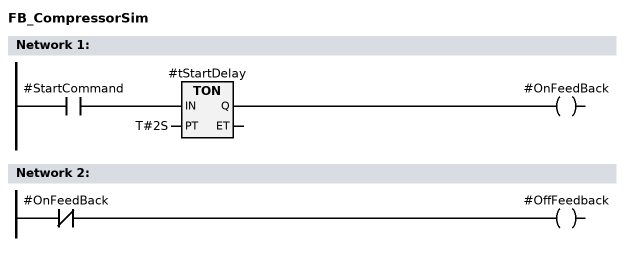
   #tStartDelay(IN := #StartCommand, PT := T#2S);   // TON
   #OnFeedBack := #tStartDelay.Q;
END_REGION

REGION Network 2
   RUNG wire#powerrail
      I_Contact( #OnFeedBack )
      Coil( #OffFeedback )
   END_RUNG
   // the same network as SCL:
   #OffFeedback := NOT #OnFeedBack;
END_REGION
END_FUNCTION_BLOCK

FUNCTION_BLOCK "FB_FanSim"   // FB9, LAD
{ S7_Optimized_Access := 'TRUE' }
VERSION : 0.1
   VAR_INPUT
      StartCommand : Bool;
   END_VAR
   VAR_OUTPUT
      OnFeedBack : Bool;
      OffFeedBack : Bool;
   END_VAR
   VAR
      tStartDelay : TON_TIME;
      SA : Bool;
   END_VAR
   VAR_TEMP
      Temp_1 : Bool;
   END_VAR
BEGIN

REGION Network 1
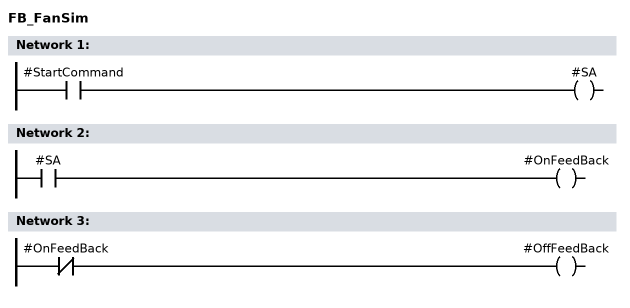
   RUNG wire#powerrail
      Contact( #StartCommand )
      Coil( #SA )
   END_RUNG
   // the same network as SCL:
   #SA := #StartCommand;
END_REGION

REGION Network 2
   RUNG wire#powerrail
      Contact( #SA )
      Coil( #OnFeedBack )
   END_RUNG
   // the same network as SCL:
   #OnFeedBack := #SA;
END_REGION

REGION Network 3
   RUNG wire#powerrail
      I_Contact( #OnFeedBack )
      Coil( #OffFeedBack )
   END_RUNG
   // the same network as SCL:
   #OffFeedBack := NOT #OnFeedBack;
END_REGION
END_FUNCTION_BLOCK

(* ===== HMI "HMI_RT_1" =====
system functions are stored by id; their names below are inferred from use
connection "HMI_Connection_1": ETHERNET, S7_1500_OMS

HMI tags "Default tag table"
   "Db_Equipment_Compressor{1}_Sts_Status" : Int = PLC Db_Equipment.Compressor[1].Sts.Status, 1 s
   "Db_Equipment_Compressor{2}_Sts_Status" : Int = PLC Db_Equipment.Compressor[2].Sts.Status, 1 s
   "Db_Equipment_Compressor{3}_Sts_Status" : Int = PLC Db_Equipment.Compressor[3].Sts.Status, 1 s
   "Db_Equipment_Compressor{4}_Sts_Status" : Int = PLC Db_Equipment.Compressor[4].Sts.Status, 1 s
   "Db_Equipment_Compressor{5}_Sts_Status" : Int = PLC Db_Equipment.Compressor[5].Sts.Status, 1 s
   "Db_Equipment_Compressor{6}_Sts_Status" : Int = PLC Db_Equipment.Compressor[6].Sts.Status, 1 s
   "Db_Equipment_Compressor{7}_Sts_Status" : Int = PLC Db_Equipment.Compressor[7].Sts.Status, 1 s
   "Db_Equipment_Compressor{8}_Sts_Status" : Int = PLC Db_Equipment.Compressor[8].Sts.Status, 1 s
   "Db_Equipment_Fan{1}_Sts_Status" : Int = PLC Db_Equipment.Fan[1].Sts.Status, 1 s
   "Db_Equipment_Fan{2}_Sts_Status" : Int = PLC Db_Equipment.Fan[2].Sts.Status, 1 s
   "Db_Equipment_Fan{3}_Sts_Status" : Int = PLC Db_Equipment.Fan[3].Sts.Status, 1 s
   "Db_Equipment_Fan{4}_Sts_Status" : Int = PLC Db_Equipment.Fan[4].Sts.Status, 1 s
   "Db_Equipment_Fan{5}_Sts_Status" : Int = PLC Db_Equipment.Fan[5].Sts.Status, 1 s
   "Db_Equipment_Fan{6}_Sts_Status" : Int = PLC Db_Equipment.Fan[6].Sts.Status, 1 s
   "Db_Equipment_Fan{7}_Sts_Status" : Int = PLC Db_Equipment.Fan[7].Sts.Status, 1 s
   "Db_Equipment_Fan{8}_Sts_Status" : Int = PLC Db_Equipment.Fan[8].Sts.Status, 1 s
   "Db_Equipment_Fan{9}_Sts_Status" : Int = PLC Db_Equipment.Fan[9].Sts.Status, 1 s
   "Db_Equipment_Fan{10}_Sts_Status" : Int = PLC Db_Equipment.Fan[10].Sts.Status, 1 s
   "Db_Equipment_Fan{11}_Sts_Status" : Int = PLC Db_Equipment.Fan[11].Sts.Status, 1 s
   "Db_Equipment_Fan{12}_Sts_Status" : Int = PLC Db_Equipment.Fan[12].Sts.Status, 1 s
   "Db_Equipment_Process_WaterTempSetPoint" : Real = PLC Db_Equipment.Process.WaterTempSetPoint, 1 s
   "Db_Equipment_Process_WaterOutletTemp" : Real = PLC Db_Equipment.Process.WaterOutletTemp, 1 s
   "Db_Equipment_Process_CompressorPercent" : Real = PLC Db_Equipment.Process.CompressorPercent, 1 s
   "Db_Equipment_Process_FanPercent" : Real = PLC Db_Equipment.Process.FanPercent, 1 s
   "DB_Machine_EnableAllEquipment" : Bool = PLC DB_Machine.EnableAllEquipment, 1 s
   "DB_Machine_DisableAllEquipment" : Bool = PLC DB_Machine.DisableAllEquipment, 1 s
   "DB_Machine_ResetAllEquipmentFaults" : Bool = PLC DB_Machine.ResetAllEquipmentFaults, 1 s
   "Db_Equipment_Compressor{1}_Cfg_Enabled" : Bool = PLC Db_Equipment.Compressor[1].Cfg.Enabled, 1 s
   "Db_Equipment_Compressor{1}_Sts_RunHours" : Real = PLC Db_Equipment.Compressor[1].Sts.RunHours, 1 s
   "Db_Equipment_Compressor{2}_Sts_RunHours" : Real = PLC Db_Equipment.Compressor[2].Sts.RunHours, 1 s
   "Db_Equipment_Compressor{3}_Sts_RunHours" : Real = PLC Db_Equipment.Compressor[3].Sts.RunHours, 1 s
   "Db_Equipment_Compressor{4}_Sts_RunHours" : Real = PLC Db_Equipment.Compressor[4].Sts.RunHours, 1 s
   "Db_Equipment_Compressor{5}_Sts_RunHours" : Real = PLC Db_Equipment.Compressor[5].Sts.RunHours, 1 s
   "Db_Equipment_Compressor{6}_Sts_RunHours" : Real = PLC Db_Equipment.Compressor[6].Sts.RunHours, 1 s
   "Db_Equipment_Compressor{7}_Sts_RunHours" : Real = PLC Db_Equipment.Compressor[7].Sts.RunHours, 1 s
   "Db_Equipment_Compressor{8}_Sts_RunHours" : Real = PLC Db_Equipment.Compressor[8].Sts.RunHours, 1 s
   "Db_Equipment_CompressorTiming_MinOnTime" : Time = PLC Db_Equipment.CompressorTiming.MinOnTime, 1 s
   "Db_Equipment_CompressorTiming_MinOffTime" : Time = PLC Db_Equipment.CompressorTiming.MinOffTime, 1 s
   "Db_Equipment_FanTiming_MinOnTime" : Time = PLC Db_Equipment.FanTiming.MinOnTime, 1 s
   "Db_Equipment_FanTiming_MinOffTime" : Time = PLC Db_Equipment.FanTiming.MinOffTime, 1 s
   "DB_Machine_LowTempLimit" : Real = PLC DB_Machine.LowTempLimit, 1 s
   "Db_Equipment_Compressor{1}_Cmd_ResetRuntime" : Bool = PLC Db_Equipment.Compressor[1].Cmd.ResetRuntime, 1 s
   "Db_Equipment_Compressor{2}_Cmd_ResetRuntime" : Bool = PLC Db_Equipment.Compressor[2].Cmd.ResetRuntime, 1 s
   "Db_Equipment_Compressor{3}_Cmd_ResetRuntime" : Bool = PLC Db_Equipment.Compressor[3].Cmd.ResetRuntime, 1 s
   "Db_Equipment_Compressor{4}_Cmd_ResetRuntime" : Bool = PLC Db_Equipment.Compressor[4].Cmd.ResetRuntime, 1 s
   "Db_Equipment_Compressor{5}_Cmd_ResetRuntime" : Bool = PLC Db_Equipment.Compressor[5].Cmd.ResetRuntime, 1 s
   "Db_Equipment_Compressor{6}_Cmd_ResetRuntime" : Bool = PLC Db_Equipment.Compressor[6].Cmd.ResetRuntime, 1 s
   "Db_Equipment_Compressor{7}_Cmd_ResetRuntime" : Bool = PLC Db_Equipment.Compressor[7].Cmd.ResetRuntime, 1 s
   "Db_Equipment_Compressor{8}_Cmd_ResetRuntime" : Bool = PLC Db_Equipment.Compressor[8].Cmd.ResetRuntime, 1 s
   "DB_Machine_StartRequest" : Bool = PLC DB_Machine.StartRequest, 1 s
   "DB_Machine_StopRequest" : Bool = PLC DB_Machine.StopRequest, 1 s
   "DB_Alarm_AlarmWord1" : Word = PLC DB_Alarm.AlarmWord1, 1 s
   "DB_Alarm_AlarmWord2" : Word = PLC DB_Alarm.AlarmWord2, 1 s
   "Db_Equipment_Process_GasPressure" : Real = PLC Db_Equipment.Process.GasPressure, 1 s
   "Db_Equipment_CompressorTiming_FeedbackTime" : Time = PLC Db_Equipment.CompressorTiming.FeedbackTime, 1 s
   "Db_Equipment_FanTiming_FeedbackTime" : Time = PLC Db_Equipment.FanTiming.FeedbackTime, 1 s

discrete alarms
   1: 'Compressor 1 - Start Feedback Fault', class Errors, trigger "DB_Alarm_AlarmWord1" bit 0
   2: 'Compressor 2 - Start Feedback Fault', class Errors, trigger "DB_Alarm_AlarmWord1" bit 1
   3: 'Compressor 3 - Start Feedback Fault', class Errors, trigger "DB_Alarm_AlarmWord1" bit 2
   4: 'Compressor 4 - Start Feedback Fault', class Errors, trigger "DB_Alarm_AlarmWord1" bit 3
   5: 'Compressor 5 - Start Feedback Fault', class Errors, trigger "DB_Alarm_AlarmWord1" bit 4
   6: 'Compressor 6 - Start Feedback Fault', class Errors, trigger "DB_Alarm_AlarmWord1" bit 5
   7: 'Compressor 7 - Start Feedback Fault', class Errors, trigger "DB_Alarm_AlarmWord1" bit 6
   8: 'Compressor 8 - Start Feedback Fault', class Errors, trigger "DB_Alarm_AlarmWord1" bit 7
   9: 'Fan 1 - Start Feedback Fault', class Errors, trigger "DB_Alarm_AlarmWord1" bit 8
   10: 'Fan 2 - Start Feedback Fault', class Errors, trigger "DB_Alarm_AlarmWord1" bit 9
   11: 'Fan 3 - Start Feedback Fault', class Errors, trigger "DB_Alarm_AlarmWord1" bit 10
   12: 'Fan 4 - Start Feedback Fault', class Errors, trigger "DB_Alarm_AlarmWord1" bit 11
   13: 'Fan 5 - Start Feedback Fault', class Errors, trigger "DB_Alarm_AlarmWord1" bit 12
   14: 'Fan 6 - Start Feedback Fault', class Errors, trigger "DB_Alarm_AlarmWord1" bit 13
   15: 'Fan 7 - Start Feedback Fault', class Errors, trigger "DB_Alarm_AlarmWord1" bit 14
   16: 'Fan 8 - Start Feedback Fault', class Errors, trigger "DB_Alarm_AlarmWord1" bit 15
   17: 'Fan 9 - Start Feedback Fault', class Errors, trigger "DB_Alarm_AlarmWord2" bit 0
   18: 'Fan 10 - Start Feedback Fault', class Errors, trigger "DB_Alarm_AlarmWord2" bit 1
   19: 'Fan 11 - Start Feedback Fault', class Errors, trigger "DB_Alarm_AlarmWord2" bit 2
   20: 'Fan 12 - Start Feedback Fault', class Errors, trigger "DB_Alarm_AlarmWord2" bit 3
   21: 'Water Flow Fault', class Errors, trigger "DB_Alarm_AlarmWord2" bit 4
   22: 'Low Temperature Alarm', class Errors, trigger "DB_Alarm_AlarmWord2" bit 5

text list "MachineStatus": 0 'Machine Off'; 1 'Machine Running'

Template "Template_1" 800x480
   Button "Template_Button_1" at 130,10 size 120x50; TextOff 'MAIN PAGE'
      on Press: ActivateScreen("main page", 0)
   Button "Template_Button_2" at 260,10 size 120x50; TextOff 'PARAMETERS'
      on Press: ActivateScreen("parametre", 0)
   Button "Template_Button_3" at 390,10 size 120x50; TextOff 'TREND'
      on Press: ActivateScreen("trend", 0)
   Button "Template_Button_4" at 520,10 size 120x50; TextOff 'ALARM'
      on Press: ActivateScreen("alarm", 0)
   TextField "Template_Text field_1" at 10,10 size 95x42; Text 'CHILLER COMPANY'
   Button "Template_Button_5" at 650,10 size 120x50; TextOff 'ALARM HISTORY'
      on Press: ActivateScreen("alarm history", 0)

screen "main page" 800x480, template "Template_1"
   TextField "Text field_1" at 46,115 size 102x21; Text 'Kompresor 1'
   TextField "Text field_2" at 46,135 size 102x21; Text 'Kompresor 2'
   TextField "Text field_3" at 46,155 size 102x21; Text 'Kompresor 3'
   TextField "Text field_4" at 46,175 size 102x21; Text 'Kompresor 4'
   TextField "Text field_5" at 46,195 size 102x21; Text 'Kompresor 5'
   TextField "Text field_6" at 46,215 size 102x21; Text 'Kompresor 6'
   TextField "Text field_7" at 46,235 size 102x21; Text 'Kompresor 7'
   TextField "Text field_8" at 46,255 size 102x21; Text 'Kompresor 8'
   TextField "Text field_9" at 219,115 size 44x21; Text 'Fan 1'
   TextField "Text field_10" at 219,135 size 44x21; Text 'Fan 2'
   TextField "Text field_11" at 219,155 size 44x21; Text 'Fan 3'
   TextField "Text field_12" at 219,175 size 44x21; Text 'Fan 4'
   TextField "Text field_13" at 219,195 size 44x21; Text 'Fan 5'
   TextField "Text field_14" at 219,215 size 44x21; Text 'Fan 6'
   TextField "Text field_15" at 219,235 size 44x21; Text 'Fan 7'
   TextField "Text field_16" at 219,255 size 44x21; Text 'Fan 8'
   TextField "Text field_17" at 219,275 size 44x21; Text 'Fan 9'
   TextField "Text field_18" at 219,295 size 54x21; Text 'Fan 10'
   TextField "Text field_19" at 219,315 size 54x21; Text 'Fan 11'
   TextField "Text field_20" at 219,335 size 54x21; Text 'Fan 12'
   Circle "ind_Comp01Status" at 27,117 size 15x15
      Appearance <- "Db_Equipment_Compressor{1}_Sts_Status"
   Circle "ind_Comp02Status" at 27,137 size 15x15
      Appearance <- "Db_Equipment_Compressor{2}_Sts_Status"
   Circle "ind_Comp03Status" at 27,157 size 15x15
      Appearance <- "Db_Equipment_Compressor{3}_Sts_Status"
   Circle "ind_Comp04Status" at 27,177 size 15x15
      Appearance <- "Db_Equipment_Compressor{4}_Sts_Status"
   Circle "ind_Comp05Status" at 27,197 size 15x15
      Appearance <- "Db_Equipment_Compressor{5}_Sts_Status"
   Circle "ind_Comp06Status" at 27,217 size 15x15
      Appearance <- "Db_Equipment_Compressor{6}_Sts_Status"
   Circle "ind_Comp07Status" at 27,237 size 15x15
      Appearance <- "Db_Equipment_Compressor{7}_Sts_Status"
   Circle "ind_Comp08Status" at 27,257 size 15x15
      Appearance <- "Db_Equipment_Compressor{8}_Sts_Status"
   Circle "ind_Fan01Status" at 200,117 size 15x15
      Appearance <- "Db_Equipment_Fan{1}_Sts_Status"
   Circle "ind_Fan02Status" at 200,137 size 15x15
      Appearance <- "Db_Equipment_Fan{2}_Sts_Status"
   Circle "ind_Fan03Status" at 200,157 size 15x15
      Appearance <- "Db_Equipment_Fan{3}_Sts_Status"
   Circle "ind_Fan04Status" at 200,177 size 15x15
      Appearance <- "Db_Equipment_Fan{4}_Sts_Status"
   Circle "ind_Fan05Status" at 200,197 size 15x15
      Appearance <- "Db_Equipment_Fan{5}_Sts_Status"
   Circle "ind_Fan06Status" at 200,217 size 15x15
      Appearance <- "Db_Equipment_Fan{6}_Sts_Status"
   Circle "ind_Fan07Status" at 200,237 size 15x15
      Appearance <- "Db_Equipment_Fan{7}_Sts_Status"
   Circle "ind_Fan09Status" at 200,258 size 15x15
      Appearance <- "Db_Equipment_Fan{8}_Sts_Status"
   Circle "ind_Fan10Status" at 200,277 size 15x15
      Appearance <- "Db_Equipment_Fan{9}_Sts_Status"
   Circle "ind_Fan12Status" at 200,317 size 15x15
      Appearance <- "Db_Equipment_Fan{11}_Sts_Status"
   Circle "ind_Fan11Status" at 200,297 size 15x15
      Appearance <- "Db_Equipment_Fan{10}_Sts_Status"
   Circle "ind_Fan12Status_1" at 200,337 size 15x15
      Appearance <- "Db_Equipment_Fan{12}_Sts_Status"
   TextField "Text field_21" at 46,377 size 31x21; Text 'OFF'
   TextField "Text field_22" at 46,397 size 25x21; Text 'ON'
   TextField "Text field_23" at 46,417 size 51x21; Text 'FAULT'
   Button "Button_1" at 306,413 size 121x44; TextOff 'MACHINE START'
      on Press: function_b14e0dd5("DB_Machine_StartRequest", 0)
   Button "Button_2" at 483,413 size 121x44; TextOff 'MACHINE STOP'
      on Press: function_b14e0dd5("DB_Machine_StopRequest", 0)
   Button "Button_3" at 662,413 size 121x44; TextOff 'ALARM RESET'
      on Press: function_b14e0dd5("DB_Machine_ResetAllEquipmentFaults", 0)
   TextField "Text field_24" at 337,121 size 179x23; Text 'Water Outlet Temp'
   TextField "Text field_25" at 575,121 size 216x23; Text 'Water Outlet Set Value'
   IOField "I/O field_1" at 338,154 size 96x32; FormatPattern 99.9
      ProcessValue <- "Db_Equipment_Process_WaterOutletTemp"
   IOField "I/O field_2" at 575,154 size 96x32; FormatPattern 99.9
      ProcessValue <- "Db_Equipment_Process_WaterTempSetPoint"
   TextField "Text field_26" at 337,216 size 221x23; Text 'Compressor Capacity %'
   TextField "Text field_27" at 575,213 size 147x23; Text 'Fan Capacity %'
   IOField "I/O field_3" at 342,245 size 96x32; FormatPattern 999
      ProcessValue <- "Db_Equipment_Process_CompressorPercent"
   IOField "I/O field_4" at 579,249 size 96x32; FormatPattern 999
      ProcessValue <- "Db_Equipment_Process_FanPercent"
   TextField "Text field_28" at 327,68 size 109x23; Text 'MAIN PAGE'
   SymbolicIOField "Symbolic I/O field_1" at 15,451 size 170x32; TextOff '0'; TextOn '1'; TextList "MachineStatus"
      ProcessValue <- "Db_Equipment_Compressor{1}_Cfg_Enabled"
      Appearance <- "Db_Equipment_Compressor{1}_Cfg_Enabled"
   TextField "Text field_29" at 337,315 size 201x23; Text 'Suction Line Pressure'
   TextField "Text field_30" at 575,312 size 209x23; Text 'Suction Line Set Value'
   IOField "I/O field_5" at 342,344 size 96x32; FormatPattern 99.9
      ProcessValue <- "Db_Equipment_Process_GasPressure"
   IOField "I/O field_6" at 579,348 size 96x32; FormatPattern 99.9
      ProcessValue <- "Db_Equipment_Process_WaterTempSetPoint"

screen "parametre" 800x480, template "Template_1"
   TextField "Text field_21" at 39,96 size 16x23; Text 'Text'
   IOField "io_CompressorRestartDelay" at 220,118 size 96x32; FormatPattern 9999
      ProcessValue <- "Db_Equipment_CompressorTiming_MinOnTime"
   TextField "Text field_1" at 450,120 size 115x21; Text 'Compressor 1'
   IOField "io_Comp01RunHours" at 570,120 size 96x32; FormatPattern 9999
      ProcessValue <- "Db_Equipment_Compressor{1}_Sts_RunHours"
   IOField "io_Comp02RunHours" at 570,150 size 96x32; FormatPattern 9999
      ProcessValue <- "Db_Equipment_Compressor{2}_Sts_RunHours"
   IOField "io_Comp03RunHours" at 570,180 size 96x32; FormatPattern 9999
      ProcessValue <- "Db_Equipment_Compressor{3}_Sts_RunHours"
   IOField "io_Comp04RunHours" at 570,210 size 96x32; FormatPattern 9999
      ProcessValue <- "Db_Equipment_Compressor{4}_Sts_RunHours"
   TextField "Text field_2" at 450,150 size 115x21; Text 'Compressor 2'
   TextField "Text field_3" at 450,180 size 110x21; Text 'Compressor 3'
   TextField "Text field_4" at 450,210 size 110x21; Text 'Compressor 4'
   TextField "Text field_5" at 130,75 size 118x23; Text 'PARAMETRE'
   Button "btn_ResetRunHours" at 574,402 size 118x49; TextOff 'TOTAL TIME RESET'
      on Press: function_b14e0dd5("Db_Equipment_Compressor{1}_Cmd_ResetRuntime", 0); function_b14e0dd5("Db_Equipment_Compressor{2}_Cmd_ResetRuntime", 0); function_b14e0dd5("Db_Equipment_Compressor{3}_Cmd_ResetRuntime", 0); function_b14e0dd5("Db_Equipment_Compressor{4}_Cmd_ResetRuntime", 0); function_b14e0dd5("Db_Equipment_Compressor{5}_Cmd_ResetRuntime", 0); function_b14e0dd5("Db_Equipment_Compressor{6}_Cmd_ResetRuntime", 0); function_b14e0dd5("Db_Equipment_Compressor{7}_Cmd_ResetRuntime", 0); function_b14e0dd5("Db_Equipment_Compressor{8}_Cmd_ResetRuntime", 0)
   TextField "Text field_6" at 450,240 size 110x21; Text 'Compressor 5'
   IOField "io_Comp01RunHours_5" at 570,240 size 96x32; FormatPattern 9999
      ProcessValue <- "Db_Equipment_Compressor{5}_Sts_RunHours"
   IOField "io_Comp02RunHours_6" at 570,270 size 96x32; FormatPattern 9999
      ProcessValue <- "Db_Equipment_Compressor{6}_Sts_RunHours"
   IOField "io_Comp03RunHours_7" at 570,300 size 96x32; FormatPattern 9999
      ProcessValue <- "Db_Equipment_Compressor{7}_Sts_RunHours"
   IOField "io_Comp04RunHours_8" at 570,330 size 96x32; FormatPattern 9999
      ProcessValue <- "Db_Equipment_Compressor{8}_Sts_RunHours"
   TextField "Text field_7" at 450,270 size 110x21; Text 'Compressor 6'
   TextField "Text field_8" at 450,300 size 110x21; Text 'Compressor 7'
   TextField "Text field_9" at 450,330 size 110x21; Text 'Compressor 8'
   TextField "Text field_10" at 25,120 size 201x21; Text 'Compressor Min On Time'
   TextField "Text field_11" at 25,150 size 203x21; Text 'Compressor Min Off Time'
   TextField "Text field_12" at 25,180 size 135x21; Text 'Fan Min On Time'
   TextField "Text field_13" at 25,210 size 137x21; Text 'Fan Min Off Time'
   IOField "io_CompressorRestartDelay_1" at 220,148 size 96x32; FormatPattern 9999
      ProcessValue <- "Db_Equipment_CompressorTiming_MinOffTime"
   IOField "io_CompressorRestartDelay_2" at 220,178 size 96x32; FormatPattern 9999
      ProcessValue <- "Db_Equipment_FanTiming_MinOnTime"
   IOField "io_CompressorRestartDelay_3" at 220,208 size 96x32; FormatPattern 9999
      ProcessValue <- "Db_Equipment_FanTiming_MinOffTime"
   TextField "Text field_14" at 41,227 size 16x23; Text 'Text'
   IOField "io_CompressorRestartDelay_4" at 220,238 size 96x32; FormatPattern s99.9
      ProcessValue <- "DB_Machine_LowTempLimit"
   TextField "Text field_15" at 25,240 size 194x21; Text 'Low Temperature Alarm'
   TextField "Text field_16" at 25,270 size 223x38; Text 'Compressor Feedback Fault Delay'
   IOField "io_CompressorRestartDelay_5" at 220,268 size 96x32; FormatPattern 9999
      ProcessValue <- "Db_Equipment_CompressorTiming_FeedbackTime"
   TextField "Text field_17" at 47,306 size 16x23; Text 'Text'
   IOField "io_CompressorRestartDelay_6" at 220,298 size 96x32; FormatPattern 9999
      ProcessValue <- "Db_Equipment_FanTiming_FeedbackTime"
   TextField "Text field_18" at 25,300 size 198x21; Text 'Fan Feedback Fault Delay'
   TextField "Text field_19" at 485,75 size 229x23; Text 'TOTAL WORKING HOURS'

screen "trend" 800x480, template "Template_1"
   TrendView "Trend view_1" at 0,75 size 799x404

screen "alarm" 800x480, template "Template_1"
   AlarmView "Alarm view_1" at 11,100 size 782x306; AlarmLog "AlarmHistory"
   Button "Button_3" at 333,413 size 137x52; TextOff 'ALARM RESET'
      on Press: function_b14e0dd5("DB_Machine_ResetAllEquipmentFaults", 0)

screen "alarm history" 800x480, template "Template_1"
   AlarmView "Alarm view_1" at 11,100 size 782x306; AlarmLog "AlarmHistory"
*)